ADAPTER IEmergencyReactorToSludgeBuffer (* Adapter Interface *)
  (* Standard: 61499-1 *)
  (* Version 0.0, 9/17/2026, Schneider Electric *)
  PACKAGE SE.Nereda;
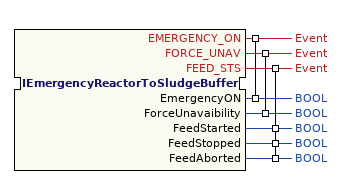
  EVENT_OUTPUT
    EMERGENCY_ON WITH EmergencyON;
    FORCE_UNAV WITH ForceUnavaibility;
    FEED_STS WITH FeedStarted, FeedStopped, FeedAborted;
  END_EVENT
  VAR_OUTPUT
    EmergencyON : BOOL;
    ForceUnavaibility : BOOL;
    FeedStarted : BOOL;
    FeedStopped : BOOL;
    FeedAborted : BOOL;
  END_VAR
  SERVICE SOCKET/PLUG
    SEQUENCE request_confirm
      SOCKET.REQ(REQD) -> PLUG.REQ(REQD);
      PLUG.CNF(CNFD) -> SOCKET.CNF(CNFD);
    END_SEQUENCE
    SEQUENCE indication_response
      PLUG.IND(INDD) -> SOCKET.IND(INDD);
      SOCKET.RSP(RSPD) -> PLUG.RSP(RSPD);
    END_SEQUENCE
  END_SERVICE
END_ADAPTER
